{attribute 'GeneratedUsingTerminal: KL3361'}
{attribute addProperty BoxType "KL3361"}
{attribute addProperty Id "StateAT %I*USINT0Data_In_0AT %I*UINT0Data_In_1AT %I*UINT0Data_In_2AT %I*UINT0Data_In_3AT %I*UINT0Data_In_4AT %I*UINT0Data_In_5AT %I*UINT0Data_In_6AT %I*UINT0Data_In_7AT %I*UINT0Data_In_8AT %I*UINT0Data_In_9AT %I*UINT0Data_In_10AT %I*UINT0CtrlAT %Q*USINT0Data_Out_0AT %Q*UINT0Data_Out_1AT %Q*UINT0Data_Out_2AT %Q*UINT0Data_Out_3AT %Q*UINT0Data_Out_4AT %Q*UINT0Data_Out_5AT %Q*UINT0Data_Out_6AT %Q*UINT0Data_Out_7AT %Q*UINT0Data_Out_8AT %Q*UINT0Data_Out_9AT %Q*UINT0Data_Out_10AT %Q*UINT0"}
{attribute addProperty CRC "2018975668"}
{attribute addProperty Size "0"}
TYPE Channel_78571FB4 :
STRUCT
	{attribute addProperty Name "State"}
	State AT %I* : USINT;
	{attribute addProperty Name "Data_In_0"}
	Data_In_0 AT %I* : UINT;
	{attribute addProperty Name "Data_In_1"}
	Data_In_1 AT %I* : UINT;
	{attribute addProperty Name "Data_In_2"}
	Data_In_2 AT %I* : UINT;
	{attribute addProperty Name "Data_In_3"}
	Data_In_3 AT %I* : UINT;
	{attribute addProperty Name "Data_In_4"}
	Data_In_4 AT %I* : UINT;
	{attribute addProperty Name "Data_In_5"}
	Data_In_5 AT %I* : UINT;
	{attribute addProperty Name "Data_In_6"}
	Data_In_6 AT %I* : UINT;
	{attribute addProperty Name "Data_In_7"}
	Data_In_7 AT %I* : UINT;
	{attribute addProperty Name "Data_In_8"}
	Data_In_8 AT %I* : UINT;
	{attribute addProperty Name "Data_In_9"}
	Data_In_9 AT %I* : UINT;
	{attribute addProperty Name "Data_In_10"}
	Data_In_10 AT %I* : UINT;
	{attribute addProperty Name "Ctrl"}
	Ctrl AT %Q* : USINT;
	{attribute addProperty Name "Data_Out_0"}
	Data_Out_0 AT %Q* : UINT;
	{attribute addProperty Name "Data_Out_1"}
	Data_Out_1 AT %Q* : UINT;
	{attribute addProperty Name "Data_Out_2"}
	Data_Out_2 AT %Q* : UINT;
	{attribute addProperty Name "Data_Out_3"}
	Data_Out_3 AT %Q* : UINT;
	{attribute addProperty Name "Data_Out_4"}
	Data_Out_4 AT %Q* : UINT;
	{attribute addProperty Name "Data_Out_5"}
	Data_Out_5 AT %Q* : UINT;
	{attribute addProperty Name "Data_Out_6"}
	Data_Out_6 AT %Q* : UINT;
	{attribute addProperty Name "Data_Out_7"}
	Data_Out_7 AT %Q* : UINT;
	{attribute addProperty Name "Data_Out_8"}
	Data_Out_8 AT %Q* : UINT;
	{attribute addProperty Name "Data_Out_9"}
	Data_Out_9 AT %Q* : UINT;
	{attribute addProperty Name "Data_Out_10"}
	Data_Out_10 AT %Q* : UINT;
END_STRUCT
END_TYPE

(* stored: Version 1.2.0.0, ProductVersion 3.1.4024.9
   DUT Channel_78571FB4: Id {55cef6d4-9715-4892-8565-9c466dbd0078} *)
